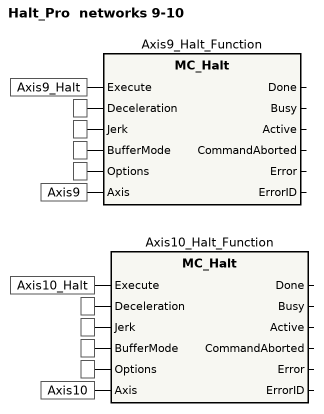
[picture p24: Halt_Pro (FBD) networks 9-10]
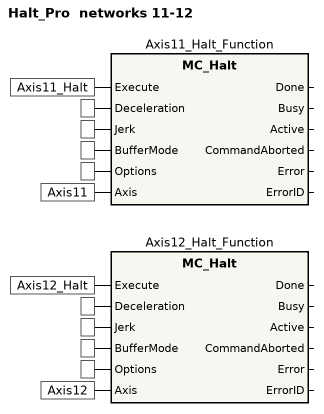
_FBD_ (* Function Block Diagram *)
NETWORK 1
	Axis1_Halt_Function:MC_Halt(Execute: Axis1_Halt, Deceleration: , Jerk: , BufferMode: , Options: , Axis: Axis1)
NETWORK 2
	Axis2_Halt_Function:MC_Halt(Execute: Axis2_Halt, Deceleration: , Jerk: , BufferMode: , Options: , Axis: Axis2)
NETWORK 3
	Axis3_Halt_Function:MC_Halt(Execute: Axis3_Halt, Deceleration: , Jerk: , BufferMode: , Options: , Axis: Axis3)
NETWORK 4
	Axis4_Halt_Function:MC_Halt(Execute: Axis4_Halt, Deceleration: , Jerk: , BufferMode: , Options: , Axis: Axis4)
NETWORK 5
	Axis5_Halt_Function:MC_Halt(Execute: Axis5_Halt, Deceleration: , Jerk: , BufferMode: , Options: , Axis: Axis5)
NETWORK 6
	Axis6_Halt_Function:MC_Halt(Execute: Axis6_Halt, Deceleration: , Jerk: , BufferMode: , Options: , Axis: Axis6)
NETWORK 7
	Axis7_Halt_Function:MC_Halt(Execute: Axis7_Halt, Deceleration: , Jerk: , BufferMode: , Options: , Axis: Axis7)
NETWORK 8
	Axis8_Halt_Function:MC_Halt(Execute: Axis8_Halt, Deceleration: , Jerk: , BufferMode: , Options: , Axis: Axis8)
NETWORK 9
	Axis9_Halt_Function:MC_Halt(Execute: Axis9_Halt, Deceleration: , Jerk: , BufferMode: , Options: , Axis: Axis9)
NETWORK 10
	Axis10_Halt_Function:MC_Halt(Execute: Axis10_Halt, Deceleration: , Jerk: , BufferMode: , Options: , Axis: Axis10)
NETWORK 11
	Axis11_Halt_Function:MC_Halt(Execute: Axis11_Halt, Deceleration: , Jerk: , BufferMode: , Options: , Axis: Axis11)
NETWORK 12
	Axis12_Halt_Function:MC_Halt(Execute: Axis12_Halt, Deceleration: , Jerk: , BufferMode: , Options: , Axis: Axis12)
_END_FBD_
END_PROGRAM

(* POU Other_Folder/Motion/Motion_Rst, LD *)
PROGRAM Motion_Rst
VAR

END_VAR
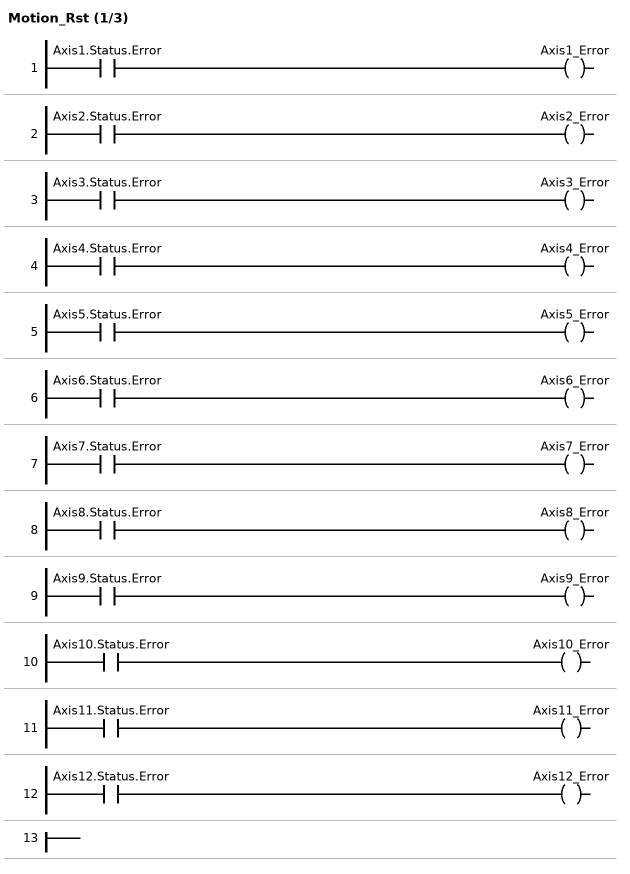
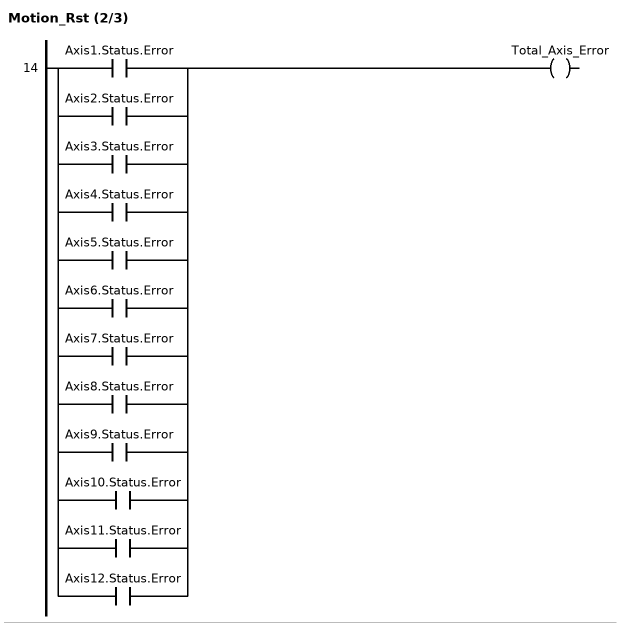
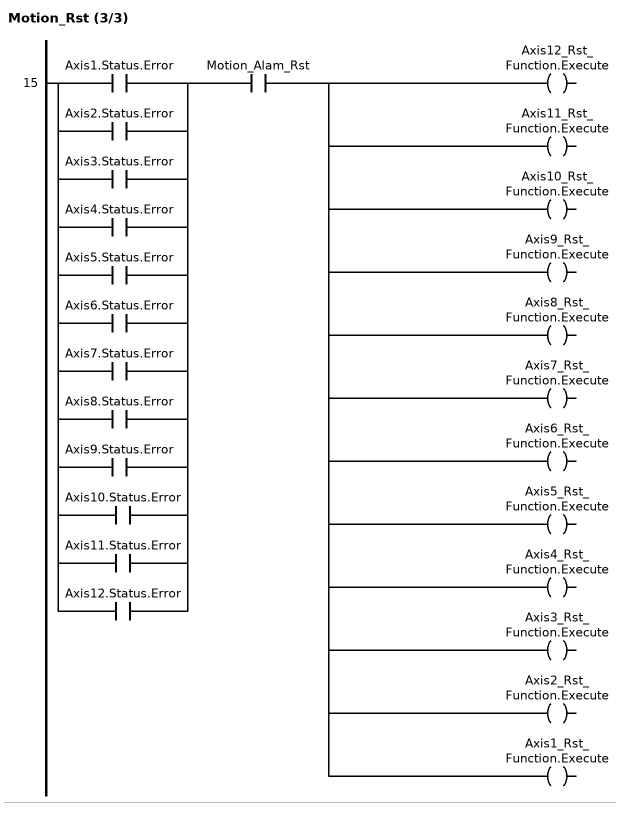
_LD_ (* Ladder Diagram *)
NETWORK 1
	[Axis1.Status.Error] --- (Axis1_Error)
NETWORK 2
	[Axis2.Status.Error] --- (Axis2_Error)
NETWORK 3
	[Axis3.Status.Error] --- (Axis3_Error)
NETWORK 4
	[Axis4.Status.Error] --- (Axis4_Error)
NETWORK 5
	[Axis5.Status.Error] --- (Axis5_Error)
NETWORK 6
	[Axis6.Status.Error] --- (Axis6_Error)
NETWORK 7
	[Axis7.Status.Error] --- (Axis7_Error)
NETWORK 8
	[Axis8.Status.Error] --- (Axis8_Error)
NETWORK 9
	[Axis9.Status.Error] --- (Axis9_Error)
NETWORK 10
	[Axis10.Status.Error] --- (Axis10_Error)
NETWORK 11
	[Axis11.Status.Error] --- (Axis11_Error)
NETWORK 12
	[Axis12.Status.Error] --- (Axis12_Error)
NETWORK 13
	*
NETWORK 14
	{ [Axis1.Status.Error] | [Axis2.Status.Error] | [Axis3.Status.Error] | [Axis4.Status.Error] | [Axis5.Status.Error] | [Axis6.Status.Error] | [Axis7.Status.Error] | [Axis8.Status.Error] | [Axis9.Status.Error] | [Axis10.Status.Error] | [Axis11.Status.Error] | [Axis12.Status.Error] } --- (Total_Axis_Error)
NETWORK 15
	{ [Axis1.Status.Error] | [Axis2.Status.Error] | [Axis3.Status.Error] | [Axis4.Status.Error] | [Axis5.Status.Error] | [Axis6.Status.Error] | [Axis7.Status.Error] | [Axis8.Status.Error] | [Axis9.Status.Error] | [Axis10.Status.Error] | [Axis11.Status.Error] | [Axis12.Status.Error] } - [Motion_Alam_Rst] --- (Axis12_Rst_Function.Execute) (Axis11_Rst_Function.Execute) (Axis10_Rst_Function.Execute) (Axis9_Rst_Function.Execute) (Axis8_Rst_Function.Execute) (Axis7_Rst_Function.Execute) (Axis6_Rst_Function.Execute) (Axis5_Rst_Function.Execute) (Axis4_Rst_Function.Execute) (Axis3_Rst_Function.Execute) (Axis2_Rst_Function.Execute) (Axis1_Rst_Function.Execute)
_END_LD_
(* the same logic as Structured Text *)
(* Network 1 *)
Axis1_Error := Axis1.Status.Error;
(* Network 2 *)
Axis2_Error := Axis2.Status.Error;
(* Network 3 *)
Axis3_Error := Axis3.Status.Error;
(* Network 4 *)
Axis4_Error := Axis4.Status.Error;
(* Network 5 *)
Axis5_Error := Axis5.Status.Error;
(* Network 6 *)
Axis6_Error := Axis6.Status.Error;
(* Network 7 *)
Axis7_Error := Axis7.Status.Error;
(* Network 8 *)
Axis8_Error := Axis8.Status.Error;
(* Network 9 *)
Axis9_Error := Axis9.Status.Error;
(* Network 10 *)
Axis10_Error := Axis10.Status.Error;
(* Network 11 *)
Axis11_Error := Axis11.Status.Error;
(* Network 12 *)
Axis12_Error := Axis12.Status.Error;
(* Network 13 *)
(* Network 14 *)
Total_Axis_Error := Axis1.Status.Error OR Axis2.Status.Error OR Axis3.Status.Error OR Axis4.Status.Error OR Axis5.Status.Error OR Axis6.Status.Error OR Axis7.Status.Error OR Axis8.Status.Error OR Axis9.Status.Error OR Axis10.Status.Error OR Axis11.Status.Error OR Axis12.Status.Error;
(* Network 15 *)
Axis12_Rst_Function.Execute := (Axis1.Status.Error OR Axis2.Status.Error OR Axis3.Status.Error OR Axis4.Status.Error OR Axis5.Status.Error OR Axis6.Status.Error OR Axis7.Status.Error OR Axis8.Status.Error OR Axis9.Status.Error OR Axis10.Status.Error OR Axis11.Status.Error OR Axis12.Status.Error) AND Motion_Alam_Rst;
Axis11_Rst_Function.Execute := Axis12_Rst_Function.Execute;
Axis10_Rst_Function.Execute := Axis12_Rst_Function.Execute;
Axis9_Rst_Function.Execute := Axis12_Rst_Function.Execute;
Axis8_Rst_Function.Execute := Axis12_Rst_Function.Execute;
Axis7_Rst_Function.Execute := Axis12_Rst_Function.Execute;
Axis6_Rst_Function.Execute := Axis12_Rst_Function.Execute;
Axis5_Rst_Function.Execute := Axis12_Rst_Function.Execute;
Axis4_Rst_Function.Execute := Axis12_Rst_Function.Execute;
Axis3_Rst_Function.Execute := Axis12_Rst_Function.Execute;
Axis2_Rst_Function.Execute := Axis12_Rst_Function.Execute;
Axis1_Rst_Function.Execute := Axis12_Rst_Function.Execute;
END_PROGRAM

(* POU Other_Folder/Motion/MotionRst_Pro, FBD *)
PROGRAM MotionRst_Pro
VAR
END_VAR
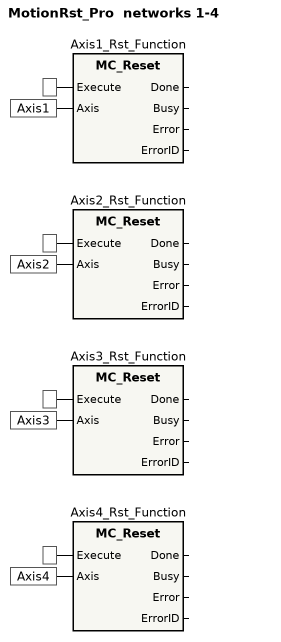
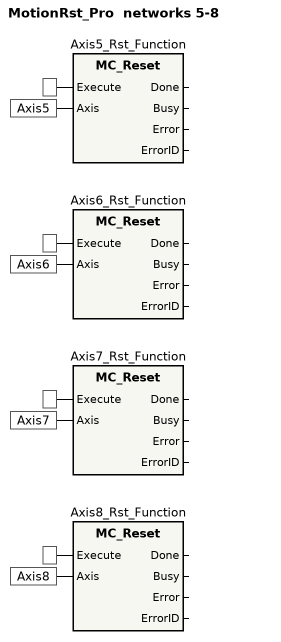
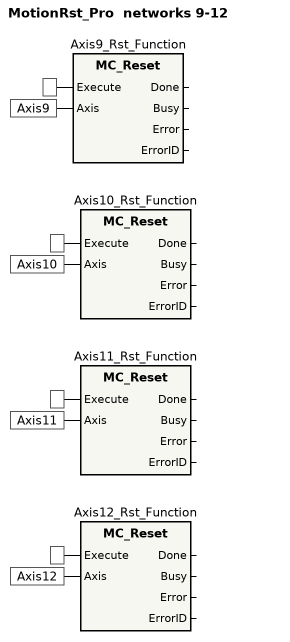
_FBD_ (* Function Block Diagram *)
NETWORK 1
	Axis1_Rst_Function:MC_Reset(Execute: , Axis: Axis1)
NETWORK 2
	Axis2_Rst_Function:MC_Reset(Execute: , Axis: Axis2)
NETWORK 3
	Axis3_Rst_Function:MC_Reset(Execute: , Axis: Axis3)
NETWORK 4
	Axis4_Rst_Function:MC_Reset(Execute: , Axis: Axis4)
NETWORK 5
	Axis5_Rst_Function:MC_Reset(Execute: , Axis: Axis5)
NETWORK 6
	Axis6_Rst_Function:MC_Reset(Execute: , Axis: Axis6)
NETWORK 7
	Axis7_Rst_Function:MC_Reset(Execute: , Axis: Axis7)
NETWORK 8
	Axis8_Rst_Function:MC_Reset(Execute: , Axis: Axis8)
NETWORK 9
	Axis9_Rst_Function:MC_Reset(Execute: , Axis: Axis9)
NETWORK 10
	Axis10_Rst_Function:MC_Reset(Execute: , Axis: Axis10)
NETWORK 11
	Axis11_Rst_Function:MC_Reset(Execute: , Axis: Axis11)
NETWORK 12
	Axis12_Rst_Function:MC_Reset(Execute: , Axis: Axis12)
_END_FBD_
END_PROGRAM

(* POU Other_Folder/Motion/PTF_Pro, FBD *)
PROGRAM PTF_Pro
VAR


END_VAR
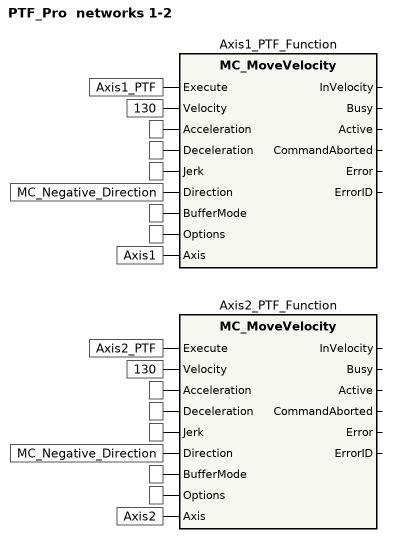
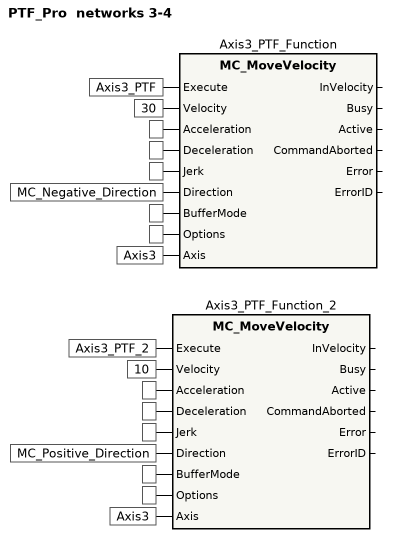
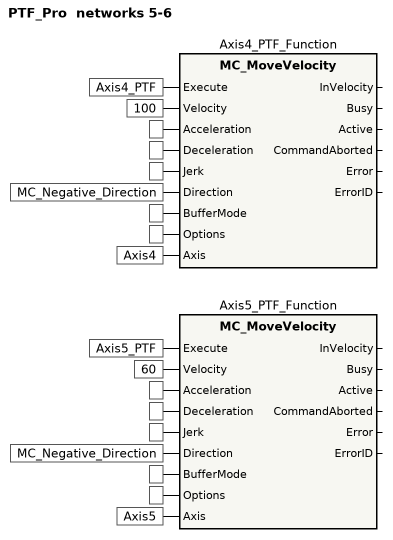
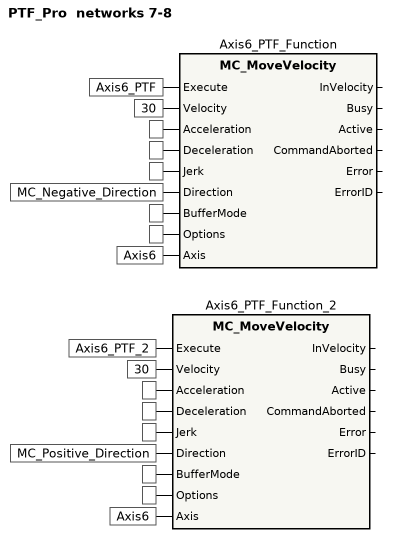
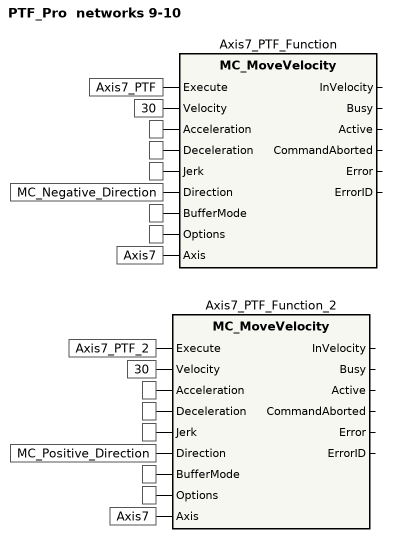
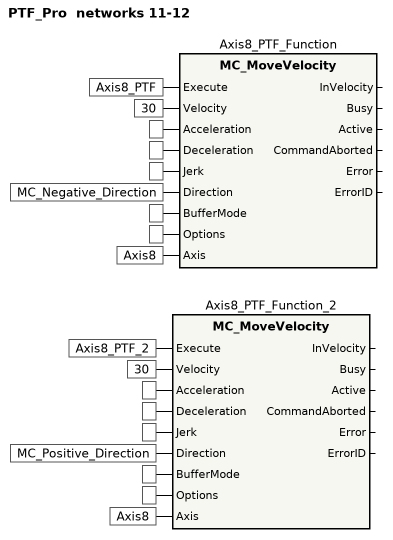
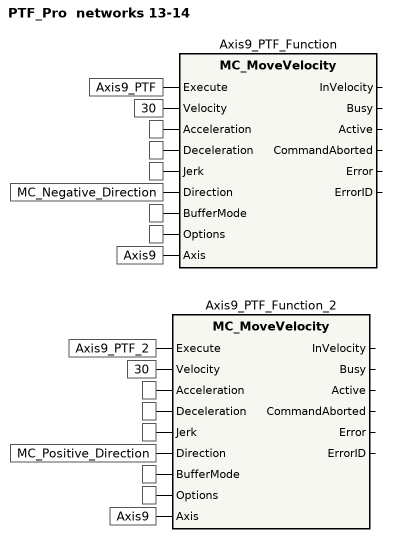
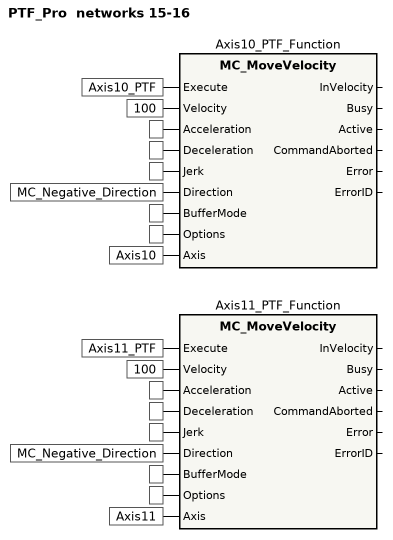
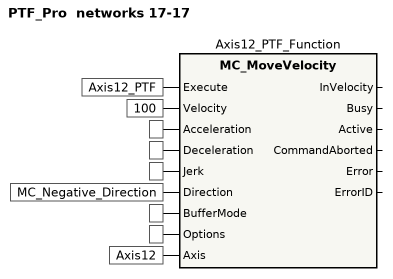
_FBD_ (* Function Block Diagram *)
NETWORK 1
	Axis1_PTF_Function:MC_MoveVelocity(Execute: Axis1_PTF, Velocity: 130, Acceleration: , Deceleration: , Jerk: , Direction: MC_Negative_Direction, BufferMode: , Options: , Axis: Axis1)
NETWORK 2
	Axis2_PTF_Function:MC_MoveVelocity(Execute: Axis2_PTF, Velocity: 130, Acceleration: , Deceleration: , Jerk: , Direction: MC_Negative_Direction, BufferMode: , Options: , Axis: Axis2)
NETWORK 3
	Axis3_PTF_Function:MC_MoveVelocity(Execute: Axis3_PTF, Velocity: 30, Acceleration: , Deceleration: , Jerk: , Direction: MC_Negative_Direction, BufferMode: , Options: , Axis: Axis3)
NETWORK 4
	Axis3_PTF_Function_2:MC_MoveVelocity(Execute: Axis3_PTF_2, Velocity: 10, Acceleration: , Deceleration: , Jerk: , Direction: MC_Positive_Direction, BufferMode: , Options: , Axis: Axis3)
NETWORK 5
	Axis4_PTF_Function:MC_MoveVelocity(Execute: Axis4_PTF, Velocity: 100, Acceleration: , Deceleration: , Jerk: , Direction: MC_Negative_Direction, BufferMode: , Options: , Axis: Axis4)
NETWORK 6
	Axis5_PTF_Function:MC_MoveVelocity(Execute: Axis5_PTF, Velocity: 60, Acceleration: , Deceleration: , Jerk: , Direction: MC_Negative_Direction, BufferMode: , Options: , Axis: Axis5)
NETWORK 7
	Axis6_PTF_Function:MC_MoveVelocity(Execute: Axis6_PTF, Velocity: 30, Acceleration: , Deceleration: , Jerk: , Direction: MC_Negative_Direction, BufferMode: , Options: , Axis: Axis6)
NETWORK 8
	Axis6_PTF_Function_2:MC_MoveVelocity(Execute: Axis6_PTF_2, Velocity: 30, Acceleration: , Deceleration: , Jerk: , Direction: MC_Positive_Direction, BufferMode: , Options: , Axis: Axis6)
NETWORK 9
	Axis7_PTF_Function:MC_MoveVelocity(Execute: Axis7_PTF, Velocity: 30, Acceleration: , Deceleration: , Jerk: , Direction: MC_Negative_Direction, BufferMode: , Options: , Axis: Axis7)
NETWORK 10
	Axis7_PTF_Function_2:MC_MoveVelocity(Execute: Axis7_PTF_2, Velocity: 30, Acceleration: , Deceleration: , Jerk: , Direction: MC_Positive_Direction, BufferMode: , Options: , Axis: Axis7)
NETWORK 11
	Axis8_PTF_Function:MC_MoveVelocity(Execute: Axis8_PTF, Velocity: 30, Acceleration: , Deceleration: , Jerk: , Direction: MC_Negative_Direction, BufferMode: , Options: , Axis: Axis8)
NETWORK 12
	Axis8_PTF_Function_2:MC_MoveVelocity(Execute: Axis8_PTF_2, Velocity: 30, Acceleration: , Deceleration: , Jerk: , Direction: MC_Positive_Direction, BufferMode: , Options: , Axis: Axis8)
NETWORK 13
	Axis9_PTF_Function:MC_MoveVelocity(Execute: Axis9_PTF, Velocity: 30, Acceleration: , Deceleration: , Jerk: , Direction: MC_Negative_Direction, BufferMode: , Options: , Axis: Axis9)
NETWORK 14
	Axis9_PTF_Function_2:MC_MoveVelocity(Execute: Axis9_PTF_2, Velocity: 30, Acceleration: , Deceleration: , Jerk: , Direction: MC_Positive_Direction, BufferMode: , Options: , Axis: Axis9)
NETWORK 15
	Axis10_PTF_Function:MC_MoveVelocity(Execute: Axis10_PTF, Velocity: 100, Acceleration: , Deceleration: , Jerk: , Direction: MC_Negative_Direction, BufferMode: , Options: , Axis: Axis10)
NETWORK 16
	Axis11_PTF_Function:MC_MoveVelocity(Execute: Axis11_PTF, Velocity: 100, Acceleration: , Deceleration: , Jerk: , Direction: MC_Negative_Direction, BufferMode: , Options: , Axis: Axis11)
NETWORK 17
	Axis12_PTF_Function:MC_MoveVelocity(Execute: Axis12_PTF, Velocity: 100, Acceleration: , Deceleration: , Jerk: , Direction: MC_Negative_Direction, BufferMode: , Options: , Axis: Axis12)
_END_FBD_
END_PROGRAM

(* POU Other_Folder/Motion/Axis_Status_Check, FBD *)
PROGRAM Axis_Status_Check
VAR
	R1: MC_ReadStatus;
	R2: MC_ReadStatus;
	R3: MC_ReadStatus;
	R4: MC_ReadStatus;
	R5: MC_ReadStatus;
	R6: MC_ReadStatus;
	R7: MC_ReadStatus;
	R8: MC_ReadStatus;
	R9: MC_ReadStatus;
	R10: MC_ReadStatus;
	R11: MC_ReadStatus;
	R12: MC_ReadStatus;
END_VAR
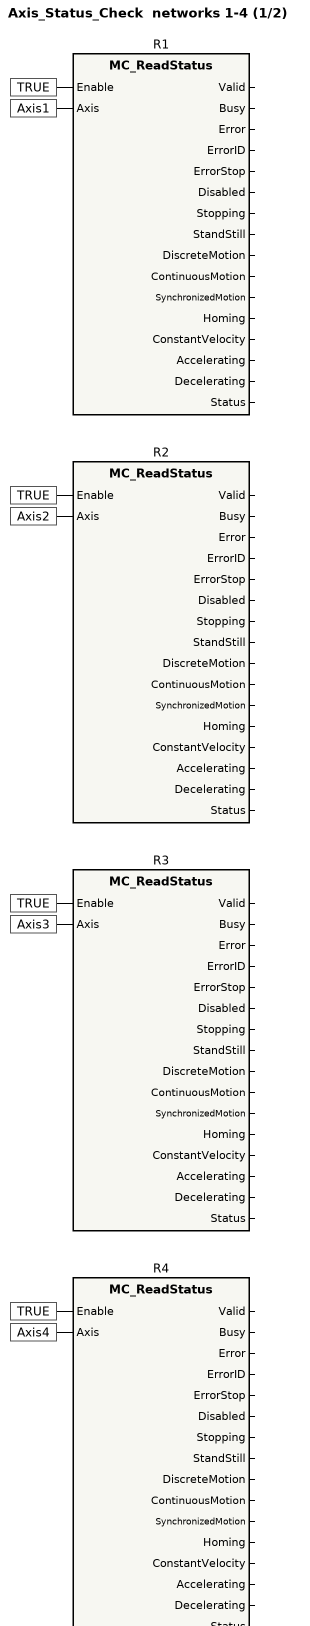
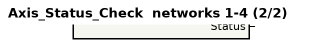
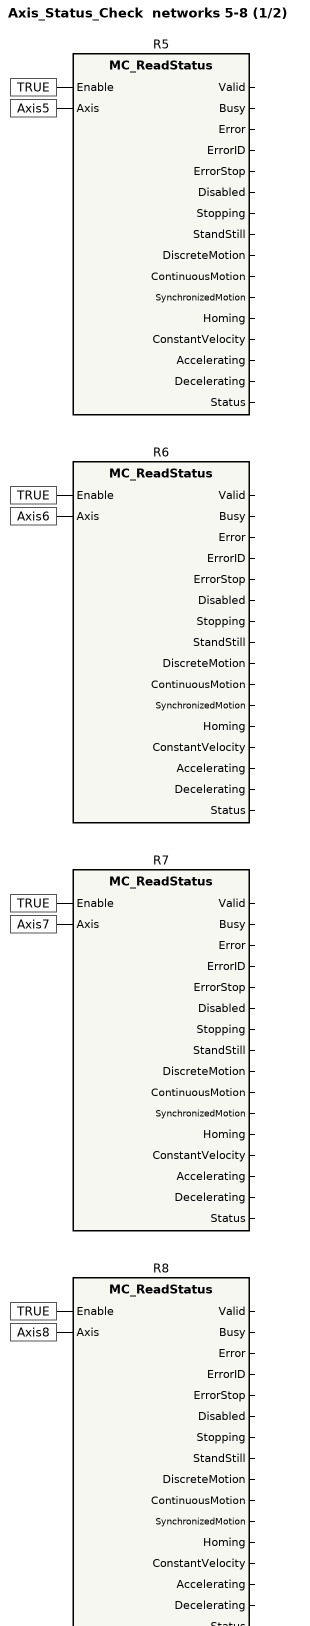
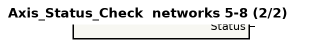
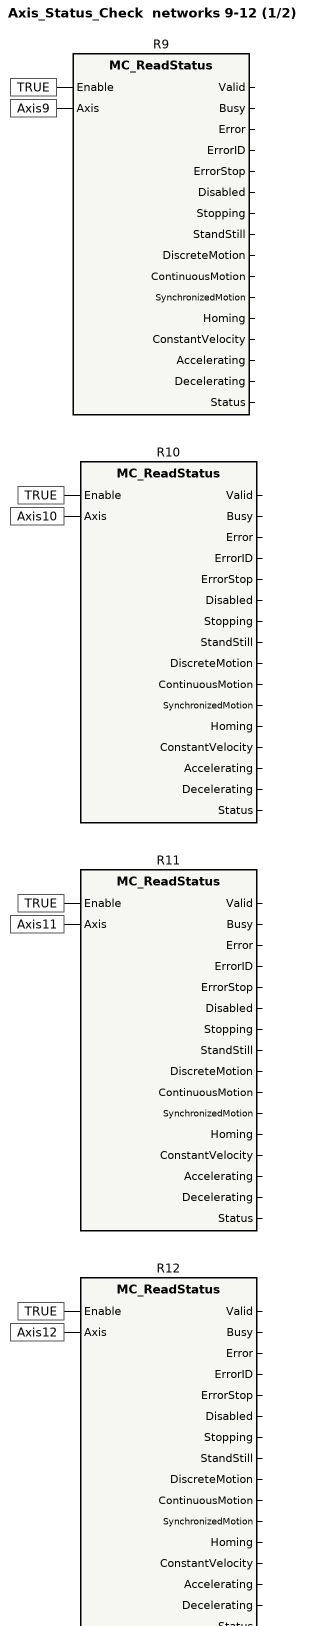
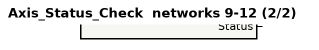
_FBD_ (* Function Block Diagram *)
NETWORK 1
	R1:MC_ReadStatus(Enable: TRUE, Axis: Axis1)
NETWORK 2
	R2:MC_ReadStatus(Enable: TRUE, Axis: Axis2)
NETWORK 3
	R3:MC_ReadStatus(Enable: TRUE, Axis: Axis3)
NETWORK 4
	R4:MC_ReadStatus(Enable: TRUE, Axis: Axis4)
NETWORK 5
	R5:MC_ReadStatus(Enable: TRUE, Axis: Axis5)
NETWORK 6
	R6:MC_ReadStatus(Enable: TRUE, Axis: Axis6)
NETWORK 7
	R7:MC_ReadStatus(Enable: TRUE, Axis: Axis7)
NETWORK 8
	R8:MC_ReadStatus(Enable: TRUE, Axis: Axis8)
NETWORK 9
	R9:MC_ReadStatus(Enable: TRUE, Axis: Axis9)
NETWORK 10
	R10:MC_ReadStatus(Enable: TRUE, Axis: Axis10)
NETWORK 11
	R11:MC_ReadStatus(Enable: TRUE, Axis: Axis11)
NETWORK 12
	R12:MC_ReadStatus(Enable: TRUE, Axis: Axis12)
_END_FBD_
(* the same logic as Structured Text *)
(* Network 1 *)
R1(Enable := TRUE, Axis := Axis1);
(* Network 2 *)
R2(Enable := TRUE, Axis := Axis2);
(* Network 3 *)
R3(Enable := TRUE, Axis := Axis3);
(* Network 4 *)
R4(Enable := TRUE, Axis := Axis4);
(* Network 5 *)
R5(Enable := TRUE, Axis := Axis5);
(* Network 6 *)
R6(Enable := TRUE, Axis := Axis6);
(* Network 7 *)
R7(Enable := TRUE, Axis := Axis7);
(* Network 8 *)
R8(Enable := TRUE, Axis := Axis8);
(* Network 9 *)
R9(Enable := TRUE, Axis := Axis9);
(* Network 10 *)
R10(Enable := TRUE, Axis := Axis10);
(* Network 11 *)
R11(Enable := TRUE, Axis := Axis11);
(* Network 12 *)
R12(Enable := TRUE, Axis := Axis12);
END_PROGRAM

(* POU Other_Folder/Speed_AxisStatus_IO/Axis_Status, LD *)
PROGRAM Axis_Status
VAR
END_VAR
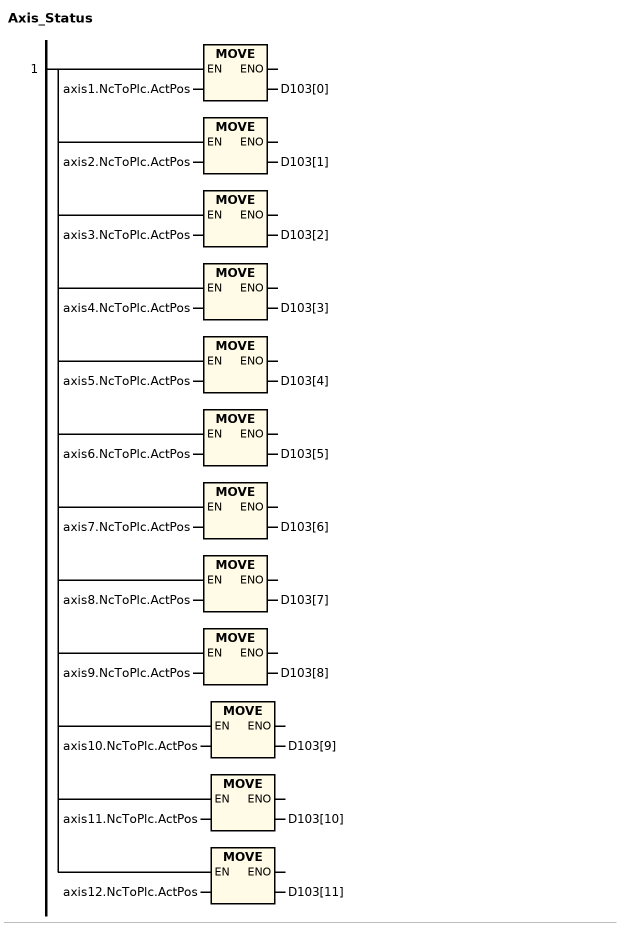
_LD_ (* Ladder Diagram *)
NETWORK 1
	*
		EN --- MOVE(axis1.NcToPlc.ActPos) => D103[0]
		EN --- MOVE(axis2.NcToPlc.ActPos) => D103[1]
		EN --- MOVE(axis3.NcToPlc.ActPos) => D103[2]
		EN --- MOVE(axis4.NcToPlc.ActPos) => D103[3]
		EN --- MOVE(axis5.NcToPlc.ActPos) => D103[4]
		EN --- MOVE(axis6.NcToPlc.ActPos) => D103[5]
		EN --- MOVE(axis7.NcToPlc.ActPos) => D103[6]
		EN --- MOVE(axis8.NcToPlc.ActPos) => D103[7]
		EN --- MOVE(axis9.NcToPlc.ActPos) => D103[8]
		EN --- MOVE(axis10.NcToPlc.ActPos) => D103[9]
		EN --- MOVE(axis11.NcToPlc.ActPos) => D103[10]
		EN --- MOVE(axis12.NcToPlc.ActPos) => D103[11]
_END_LD_
(* the same logic as Structured Text *)
(* Network 1 *)
D103[0] := axis1.NcToPlc.ActPos;
D103[1] := axis2.NcToPlc.ActPos;
D103[2] := axis3.NcToPlc.ActPos;
D103[3] := axis4.NcToPlc.ActPos;
D103[4] := axis5.NcToPlc.ActPos;
D103[5] := axis6.NcToPlc.ActPos;
D103[6] := axis7.NcToPlc.ActPos;
D103[7] := axis8.NcToPlc.ActPos;
D103[8] := axis9.NcToPlc.ActPos;
D103[9] := axis10.NcToPlc.ActPos;
D103[10] := axis11.NcToPlc.ActPos;
D103[11] := axis12.NcToPlc.ActPos;
END_PROGRAM

(* POU Other_Folder/Speed_AxisStatus_IO/Limit_Mapping, LD *)
PROGRAM Limit_Mapping
VAR

END_VAR
